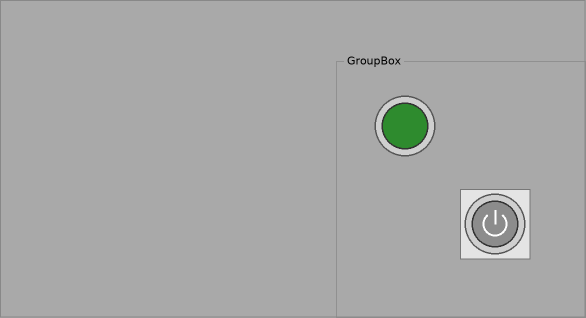
VISUALIZATION HMI  // 586x318
    GroupBox (336,53 250x265), "GroupBox"
        Lamp1 (34,38 70x70), variable: MAIN.bEnable, style: Lamp-Lamp1-Green
        PowerSwitch (124,136 70x70), variable: MAIN.bStart, behaviour: TOGGLE, style: Switch-PowerSwitch-Gray
END_VISUALIZATION

(* stored: Version 1.1.0.1, ProductVersion 3.1.4024.12
   Visu HMI: Id {fec173bc-67b0-4c63-9ff3-7bbedb99ec44} *)
